// TIA Portal V20 export
TYPE "LAxisCtrl_typeFastStop"
TITLE = LAxisCtrl_typeFastStop
// Support: tech.team.motioncontrol@siemens.com 
// Fax: +49 (0) 9131/98-1297
   STRUCT
      deceleration : LReal := -1.0;   // Deceleration for fast stop (Value > 0.0: The specified value is used; Value <= 0.0: emergency deceleration of the technology object is used)
      jerk : LReal := -1.0;   // Jerk for fast stop (Value > 0.0: Smooth velocity profile, the specified value is used; Value = 0.0: Trapezoid velocity profile; Value < 0.0: Use of the default value configured in the technology object)
      abortAcceleration : Bool := FALSE;   // TRUE: The acceleration is set to 0.0 at the start of the job, and the deceleration immediately builds up; FALSE: The current acceleration at the start of the job is reduced using the configured jerk. Afterwards, the deceleration builds up
      replaceStopPossible : Bool := FALSE;   // TRUE: Fast stop command can be replaced by another command
   END_STRUCT;
END_TYPE
